// Mitsubishi GX Works2 project: IELET2103_Oving2   PLC: FX2N/FX2NC
// IELET2103_Oving2

// task Task_01 (event TRUE, interval 0, priority 31): Oppgave1a)ST

PROGRAM Oppgave1a)ST
VAR
  tmp1 : BOOL;
END_VAR
tmp1	:=	 X0 OR (NOT X1 AND M0) AND (M0<>X0) OR NOT M1;

M0 := tmp1; 
M1 :=	tmp1 AND X1;
END_PROGRAM

PROGRAM Oppgave1a)IL
// body in language c0 not rendered
END_PROGRAM

PROGRAM Oppgave1a)LD
(* structured ladder/FBD written out as ST: instructions are called as NAME(EN, inputs, outputs); _pN, _eN, _tN stand for wires *)
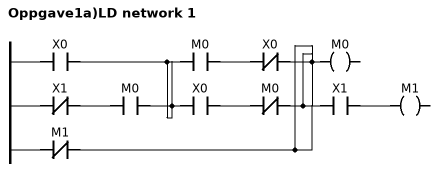
(* network 1 *)
_p1 := X0 OR (NOT X1 AND M0);
_p2 := (_p1 AND M0 AND NOT X0) OR (_p1 AND X0 AND NOT M0) OR (NOT M1);
M0 := _p2;
M1 := _p2 AND X1;
END_PROGRAM
